// TIA Portal V17 export
// export: Created 2024-08-07T21:44:09.1458819Z, ExportSetting WithDefaults, DisplayName Totally Integrated Automation Portal, DisplayVersion V17 Update 7, DisplayName TIA Portal Openness, DisplayVersion V17 Update 7, DisplayName TIA Portal Version Control Interface, DisplayVersion V17, DisplayName SINAMICS Startdrive Advanced, DisplayVersion V17 SP2, DisplayName SINAMICS Startdrive G110M, G120, G120C, G120D, G120P, G115D, DisplayVersion V17 SP2, DisplayName SINAMICS Startdrive G130, G150, S120, S150, SINAMICS MV, S210, DisplayVersion V17 SP2, DisplayName STEP 7 Professional, DisplayVersion V17 Update 7, DisplayName STEP 7 Safety, DisplayVersion V17 Update 6, DisplayName WinCC Advanced / Unified PC, DisplayVersion V17 Update 7
FUNCTION_BLOCK "FB_IJC_AWAKE_SIGNAL"   // FB1003, LAD
TITLE = Awake signal
{ S7_Optimized_Access := 'TRUE' }
VERSION : 0.1
// This function supervise Awake signal, 
// - Awake signal is to test communication between PLC and IJCORE. 
// - Awake signal is set to 1 by PLC and set to -1 by IJCORE alternatively.
// - first PLC check if awake signal is different of 1, if it is, PLC launch timer T1 
//  (1s<T1<10s). at the end of this temporisation, PLC set awake signal to 1 and 
//  launch Timer 2. 
// - if IJCORE don't set awake signal to -1 before the end of timer 2,PLC generate  
//   Time out fault for awake signal.
// stored: AutoNumber false, IsIECCheckEnabled false, IsRetainMemResEnabled false, MemoryReserve 100, SetENOAutomatically false, UDAEnableTagReadback false
   VAR_INPUT
      ack_error : Bool;
   END_VAR
   VAR_OUTPUT
      State_com : SInt;
   END_VAR
   VAR
      T1PresetValue : Time := T#1S;
      T2PresetValue : Time := T#60S;
      AwSignalTimeOutFault : Bool := 0;
      Reset_Counters : Bool;
      Restart_Counter_bit_of_life : USInt := 0;
      NB_Bit_of_Life : Bool;
      number_restart : DInt;
      check_restart : Bool;
      "Timer" { ExternalAccessible := 'False'; ExternalVisible := 'False'; ExternalWritable := 'False'} : Array[1..5] of TON_TIME;
   END_VAR
   VAR CONSTANT
      Trestart : Time := T#200ms;
      T3 : Time := T#2s;
   END_VAR
   VAR_TEMP   // added for the SCL form of the ladder/FBD networks
      _w1 : Bool;
   END_VAR
BEGIN

REGION Network 1: - if awake signal is -1 then launch timer 1
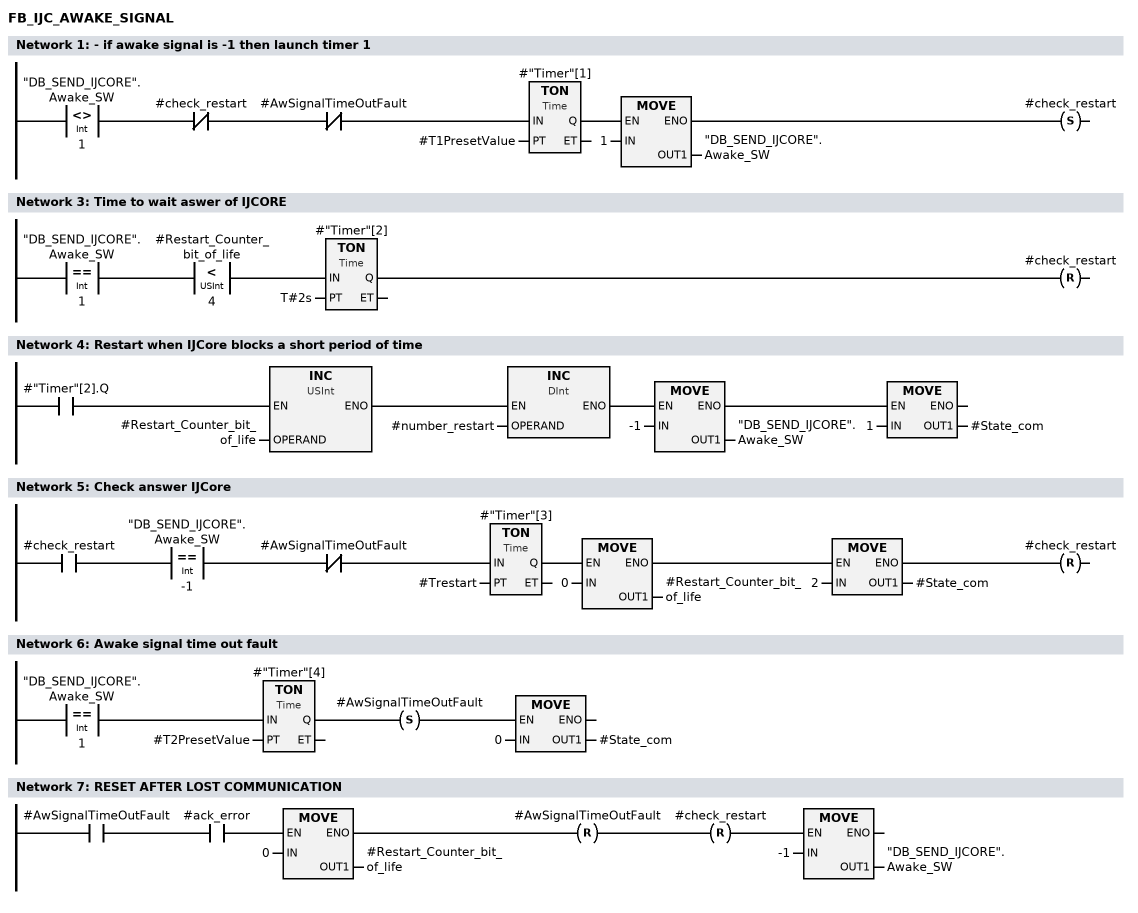
   RUNG wire#powerrail
      { S7_Templates := "SrcType := Int" } NE_Contact(in1 := "DB_SEND_IJCORE".Awake_SW, in2 := 1)
      I_Contact( #check_restart )
      I_Contact( #AwSignalTimeOutFault )
      { S7_Templates := "time_type := Time" } #"Timer"[1].TON(pt := #T1PresetValue, et =>)
      Move(in := 1, out1 => "DB_SEND_IJCORE".Awake_SW)
      S_Coil( #check_restart )
   END_RUNG
   // the same network as SCL:
   #"Timer"[1].TON(IN := ("DB_SEND_IJCORE".Awake_SW <> 1) AND NOT #check_restart AND NOT #AwSignalTimeOutFault,
                   PT := #T1PresetValue);
   IF #"Timer"[1].Q THEN
       "DB_SEND_IJCORE".Awake_SW := 1;
       #check_restart := TRUE;
   END_IF;
END_REGION

REGION Network 2: Diagnostic
END_REGION

REGION Network 3: Time to wait aswer of IJCORE
   RUNG wire#powerrail
      { S7_Templates := "SrcType := Int" } EQ_Contact(in1 := "DB_SEND_IJCORE".Awake_SW, in2 := 1)
      { S7_Templates := "SrcType := USInt" } LT_Contact(in1 := #Restart_Counter_bit_of_life, in2 := 4)
      { S7_Templates := "time_type := Time" } #"Timer"[2].TON(pt := T#2s, et =>)
      R_Coil( #check_restart )
   END_RUNG
   // the same network as SCL:
   #"Timer"[2].TON(IN := ("DB_SEND_IJCORE".Awake_SW = 1) AND (#Restart_Counter_bit_of_life < 4), PT := T#2s);
   IF #"Timer"[2].Q THEN #check_restart := FALSE; END_IF;
END_REGION

REGION Network 4: Restart when IJCore blocks a short period of time
   RUNG wire#powerrail
      Contact( #"Timer"[2].Q )
      { S7_Templates := "DestType := USInt" } Inc( #Restart_Counter_bit_of_life )
      { S7_Templates := "DestType := DInt" } Inc( #number_restart )
      Move(in := -1, out1 => "DB_SEND_IJCORE".Awake_SW)
      Move(in := 1, out1 => #State_com)
   END_RUNG
   // the same network as SCL:
   IF #"Timer"[2].Q THEN
       #Restart_Counter_bit_of_life := #Restart_Counter_bit_of_life + 1;
       #number_restart := #number_restart + 1;
       "DB_SEND_IJCORE".Awake_SW := -1;
       #State_com := 1;
   END_IF;
END_REGION

REGION Network 5: Check answer IJCore
   RUNG wire#powerrail
      Contact( #check_restart )
      { S7_Templates := "SrcType := Int" } EQ_Contact(in1 := "DB_SEND_IJCORE".Awake_SW, in2 := -1)
      I_Contact( #AwSignalTimeOutFault )
      { S7_Templates := "time_type := Time" } #"Timer"[3].TON(pt := #Trestart, et =>)
      Move(in := 0, out1 => #Restart_Counter_bit_of_life)
      Move(in := 2, out1 => #State_com)
      R_Coil( #check_restart )
   END_RUNG
   // the same network as SCL:
   #"Timer"[3].TON(IN := #check_restart AND ("DB_SEND_IJCORE".Awake_SW = (-1)) AND NOT #AwSignalTimeOutFault,
                   PT := #Trestart);
   IF #"Timer"[3].Q THEN
       #Restart_Counter_bit_of_life := 0;
       #State_com := 2;
       #check_restart := FALSE;
   END_IF;
END_REGION

REGION Network 6: Awake signal time out fault
   RUNG wire#powerrail
      { S7_Templates := "SrcType := Int" } EQ_Contact(in1 := "DB_SEND_IJCORE".Awake_SW, in2 := 1)
      { S7_Templates := "time_type := Time" } #"Timer"[4].TON(pt := #T2PresetValue, et =>)
      S_Coil( #AwSignalTimeOutFault )
      Move(in := 0, out1 => #State_com)
   END_RUNG
   // the same network as SCL:
   #"Timer"[4].TON(IN := "DB_SEND_IJCORE".Awake_SW = 1, PT := #T2PresetValue);
   IF #"Timer"[4].Q THEN
       #AwSignalTimeOutFault := TRUE;
       #State_com := 0;
   END_IF;
END_REGION

REGION Network 7: RESET AFTER LOST COMMUNICATION
   RUNG wire#powerrail
      Contact( #AwSignalTimeOutFault )
      Contact( #ack_error )
      Move(in := 0, out1 => #Restart_Counter_bit_of_life)
      R_Coil( #AwSignalTimeOutFault )
      R_Coil( #check_restart )
      Move(in := -1, out1 => "DB_SEND_IJCORE".Awake_SW)
   END_RUNG
   // the same network as SCL:
   IF #AwSignalTimeOutFault AND #ack_error THEN #Restart_Counter_bit_of_life := 0; END_IF;
   #_w1 := #AwSignalTimeOutFault AND #ack_error;
   IF #_w1 THEN
       #AwSignalTimeOutFault := FALSE;
       #check_restart := FALSE;
       "DB_SEND_IJCORE".Awake_SW := -1;
   END_IF;
END_REGION
END_FUNCTION_BLOCK
